DATA_BLOCK "AutoProcessDataPopUp_DB"
{ S7_Optimized_Access := 'TRUE' }
VERSION : 0.1
NON_RETAIN
"AutoProcessDataPopUp"

BEGIN

END_DATA_BLOCK

